{attribute 'qualified_only'}
TYPE E_JXCE1_MovementMode :
(
	ABSOLUTE := 1,
	INCREMENTAL := 2
);
END_TYPE

(* stored: Version 1.1.0.1, ProductVersion 3.1.4024.15
   DUT E_JXCE1_MovementMode: Id {38dfc45a-1daa-4656-9442-97c746252c60} *)
